Staubli VAL3: onF8Event.pgx

program onF8Event(bool& x_bSave[])
  local num l_nSize
  local tool l_tEmpty
begin
  // look if the bButton is enable
  if bButton[7]
    //
    l_tEmpty=flange
    call tcp:new(l_tEmpty.trsf)
    call tcp:getSize(l_nSize)
    nIndexTool=l_nSize-1
    // refresh and modify the name
    call buildList()
    call refreshStatic()
    nIndex=0
    sEvent=""
    call editTool(l_tEmpty)
    logMsg("[KERNEL] INTERFACE:Insert new tool at index: "+toString("",l_nSize))
    x_bSave=true
  endIf
end
